// TIA Portal V18 export
// export: Created 2026-04-18T00:00:00Z, ExportSetting WithDefaults
ORGANIZATION_BLOCK "Cyclic interrupt"   // OB30, LAD, CyclicInterrupt
{ S7_Optimized_Access := 'TRUE' }
VERSION : 0.1
// stored: AutoNumber true, IsIECCheckEnabled false
   VAR_INPUT
      Initial_Call : Bool;
      Remanence : Bool;
   END_VAR
BEGIN

REGION Network 1: Điều khiển PID
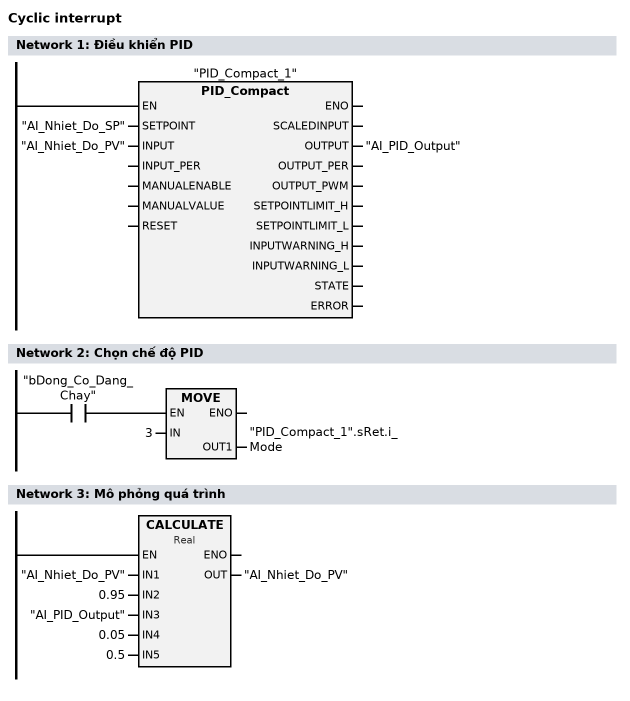
   RUNG wire#powerrail
      "PID_Compact_1".PID_Compact(Setpoint := "AI_Nhiet_Do_SP", Input := "AI_Nhiet_Do_PV", Input_PER :=, ManualEnable :=, ManualValue :=, Reset :=, ScaledInput =>, Output => "AI_PID_Output", Output_PER =>, Output_PWM =>, SetpointLimit_H =>, SetpointLimit_L =>, InputWarning_H =>, InputWarning_L =>, State =>, Error =>)
   END_RUNG
   // the same network as SCL:
   "PID_Compact_1"(Setpoint := "AI_Nhiet_Do_SP", Input := "AI_Nhiet_Do_PV", Output => "AI_PID_Output");   // PID_Compact
END_REGION

REGION Network 2: Chọn chế độ PID
   RUNG wire#powerrail
      Contact( "bDong_Co_Dang_Chay" )
      { S7_GenerateENO := "TRUE" } Move(in := 3, out1 => "PID_Compact_1".sRet.i_Mode)
   END_RUNG
   // the same network as SCL:
   IF "bDong_Co_Dang_Chay" THEN "PID_Compact_1".sRet.i_Mode := 3; END_IF;
END_REGION

REGION Network 3: Mô phỏng quá trình
   RUNG wire#powerrail
      { S7_Templates := "SrcType := Real"; S7_GenerateENO := "TRUE"; S7_Expression := "IN2*IN1 + IN4*(IN3*IN5)" } Calculate(in1 := "AI_Nhiet_Do_PV", in2 := 0.95, in3 := "AI_PID_Output", in4 := 0.05, in5 := 0.5, out => "AI_Nhiet_Do_PV")
   END_RUNG
   // the same network as SCL:
   "AI_Nhiet_Do_PV" := 0.95*"AI_Nhiet_Do_PV" + 0.05*("AI_PID_Output"*0.5);
END_REGION
END_ORGANIZATION_BLOCK
